(* Logix 5000 project; controller SX_V040001_C001 vendor 1 type 14 code 77 rev 16.23; software revision 16.04; part 30 of 35 *)
(* tags used below, declared in another part *)
   ALL_KINDS : INT[90];
   Basic : INT;
   DRIVE : INT[32];
   DRIVE_INTERVAL : INT[8];
   EMPTYING : INT[18];
   loading : INT[19];
   METERING : INT[44];
   NOTDOS : INT[6];
   pointer_recipe : DINT;
   pointer_recipe_line : DINT;
   pointer_recipe_restart : DINT;
   pointer_recipe_test : DINT;
   RECIPE_GENERAL : INT[405];
   T_MIN_ACTION_TIME : TIMER;
   TEMP : INT[14];
(* MainProgram, continued *)

ROUTINE RecipeRestart   (* ladder *)
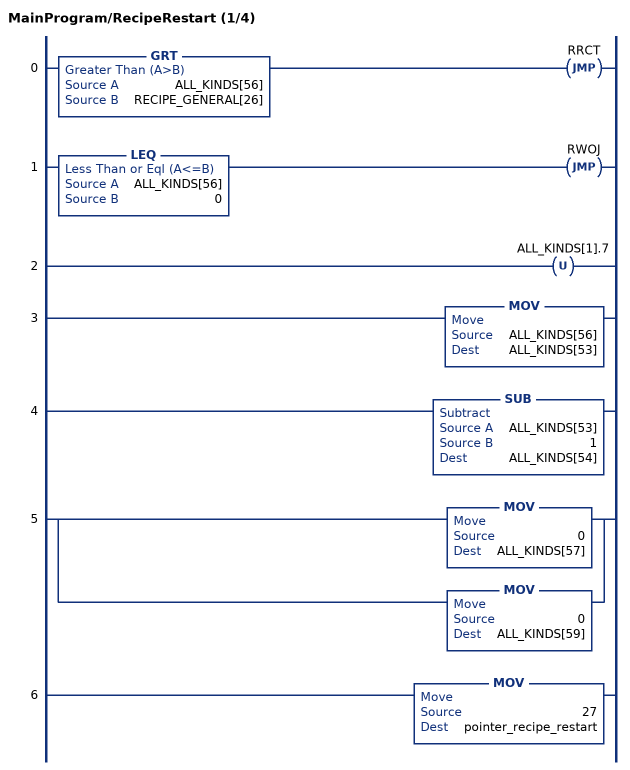
   0: GRT(ALL_KINDS[56],RECIPE_GENERAL[26])JMP(RRCT);
   1: LEQ(ALL_KINDS[56],0)JMP(RWOJ);
   2: OTU(ALL_KINDS[1].7);
   3: MOV(ALL_KINDS[56],ALL_KINDS[53]);
   4: SUB(ALL_KINDS[53],1,ALL_KINDS[54]);
   5: [MOV(0,ALL_KINDS[57]) ,MOV(0,ALL_KINDS[59]) ];
   6: MOV(27,pointer_recipe_restart);
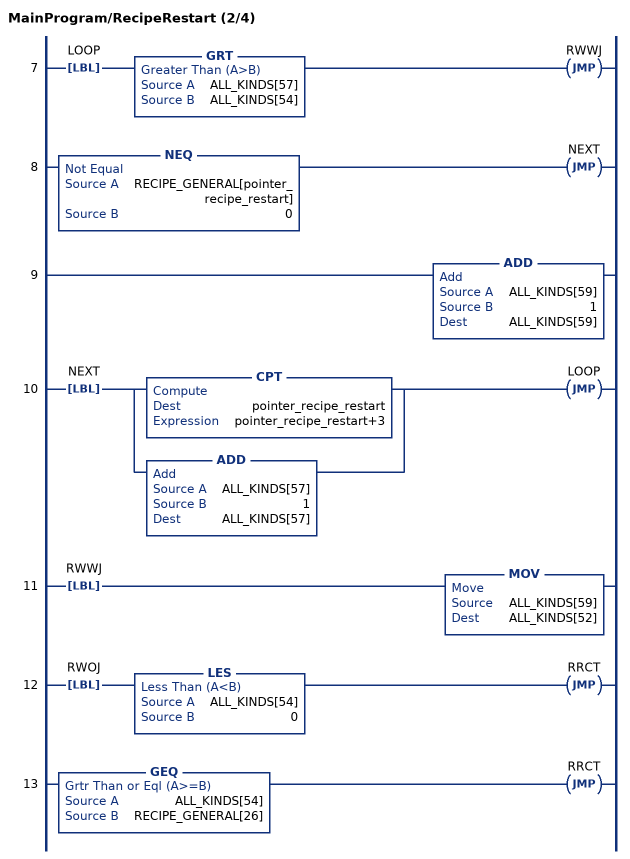
   7: LBL(LOOP)GRT(ALL_KINDS[57],ALL_KINDS[54])JMP(RWWJ);
   8: NEQ(RECIPE_GENERAL[pointer_recipe_restart],0)JMP(NEXT);
   9: ADD(ALL_KINDS[59],1,ALL_KINDS[59]);
   10: LBL(NEXT)[CPT(pointer_recipe_restart,pointer_recipe_restart+3) ,ADD(ALL_KINDS[57],1,ALL_KINDS[57]) ]JMP(LOOP);
   11: LBL(RWWJ)MOV(ALL_KINDS[59],ALL_KINDS[52]);
   12: LBL(RWOJ)LES(ALL_KINDS[54],0)JMP(RRCT);
   13: GEQ(ALL_KINDS[54],RECIPE_GENERAL[26])JMP(RRCT);
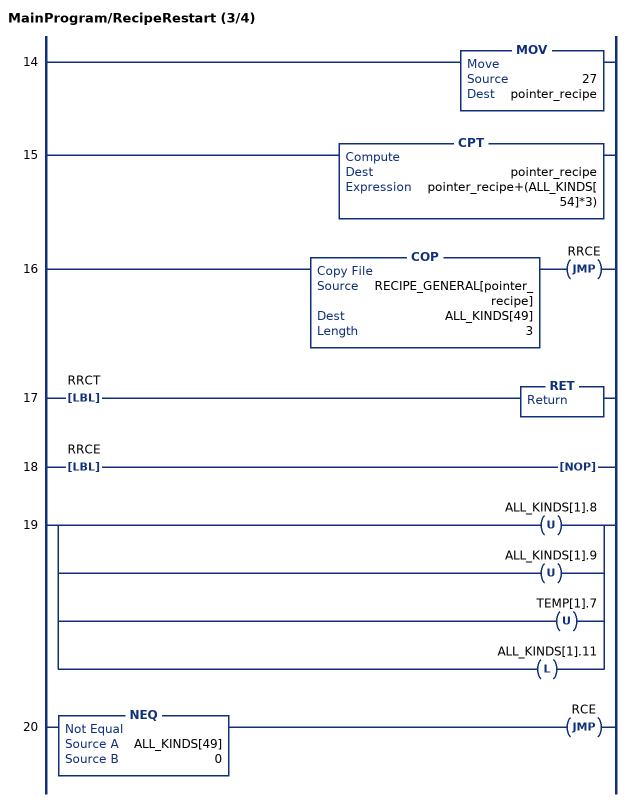
   14: MOV(27,pointer_recipe);
   15: CPT(pointer_recipe,pointer_recipe+(ALL_KINDS[54]*3));
   16: COP(RECIPE_GENERAL[pointer_recipe],ALL_KINDS[49],3)JMP(RRCE);
   17: LBL(RRCT)RET();
   18: LBL(RRCE)NOP();
   19: [OTU(ALL_KINDS[1].8) ,OTU(ALL_KINDS[1].9) ,OTU(TEMP[1].7) ,OTL(ALL_KINDS[1].11) ];
   20: NEQ(ALL_KINDS[49],0)JMP(RCE);
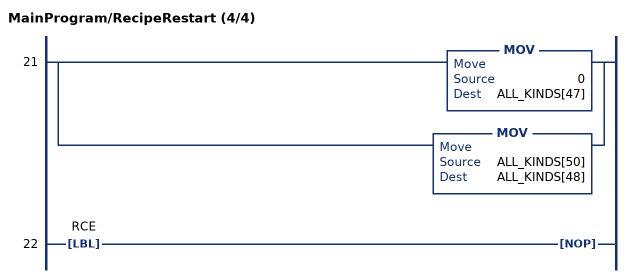
   21: [MOV(0,ALL_KINDS[47]) ,MOV(ALL_KINDS[50],ALL_KINDS[48]) ];
   22: LBL(RCE)NOP();
END_ROUTINE

ROUTINE RecipeRunning   (* ladder *)
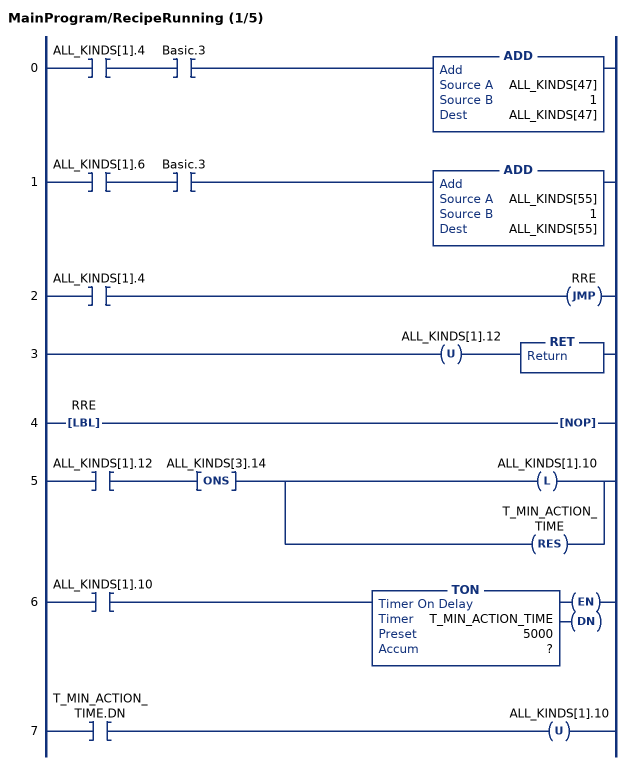
   0: XIC(ALL_KINDS[1].4)XIC(Basic.3)ADD(ALL_KINDS[47],1,ALL_KINDS[47]);
   1: XIC(ALL_KINDS[1].6)XIC(Basic.3)ADD(ALL_KINDS[55],1,ALL_KINDS[55]);
   2: XIC(ALL_KINDS[1].4)JMP(RRE);
   3: OTU(ALL_KINDS[1].12)RET();
   4: LBL(RRE)NOP();
   5: XIC(ALL_KINDS[1].12)ONS(ALL_KINDS[3].14)[OTL(ALL_KINDS[1].10) ,RES(T_MIN_ACTION_TIME) ];
   6: XIC(ALL_KINDS[1].10)TON(T_MIN_ACTION_TIME,?,?);
   7: XIC(T_MIN_ACTION_TIME.DN)OTU(ALL_KINDS[1].10);
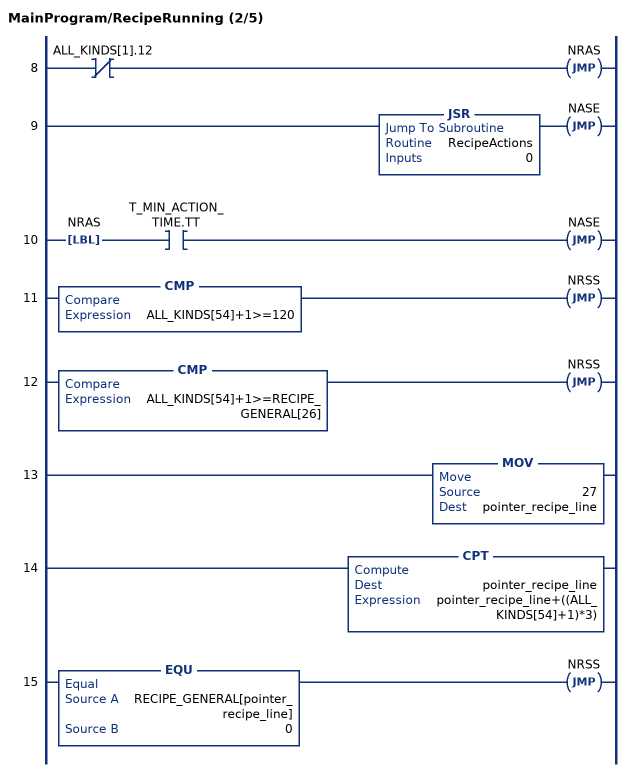
   8: XIO(ALL_KINDS[1].12)JMP(NRAS);
   9: JSR(RecipeActions,0)JMP(NASE);
   10: LBL(NRAS)XIC(T_MIN_ACTION_TIME.TT)JMP(NASE);
   11: CMP(ALL_KINDS[54]+1>=120)JMP(NRSS);
   12: CMP(ALL_KINDS[54]+1>=RECIPE_GENERAL[26])JMP(NRSS);
   13: MOV(27,pointer_recipe_line);
   14: CPT(pointer_recipe_line,pointer_recipe_line+((ALL_KINDS[54]+1)*3));
   15: EQU(RECIPE_GENERAL[pointer_recipe_line],0)JMP(NRSS);
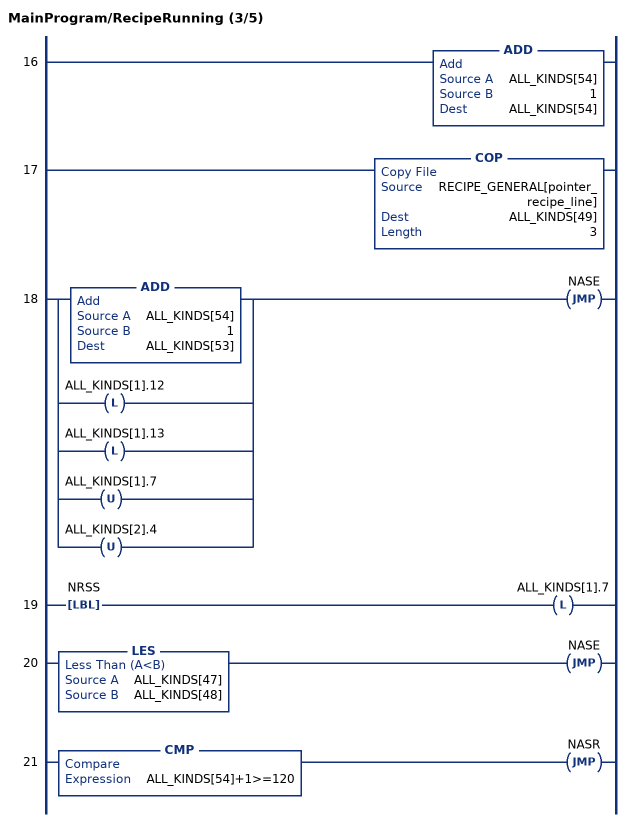
   16: ADD(ALL_KINDS[54],1,ALL_KINDS[54]);
   17: COP(RECIPE_GENERAL[pointer_recipe_line],ALL_KINDS[49],3);
   18: [ADD(ALL_KINDS[54],1,ALL_KINDS[53]) ,OTL(ALL_KINDS[1].12) ,OTL(ALL_KINDS[1].13) ,OTU(ALL_KINDS[1].7) ,OTU(ALL_KINDS[2].4) ]JMP(NASE);
   19: LBL(NRSS)OTL(ALL_KINDS[1].7);
   20: LES(ALL_KINDS[47],ALL_KINDS[48])JMP(NASE);
   21: CMP(ALL_KINDS[54]+1>=120)JMP(NASR);
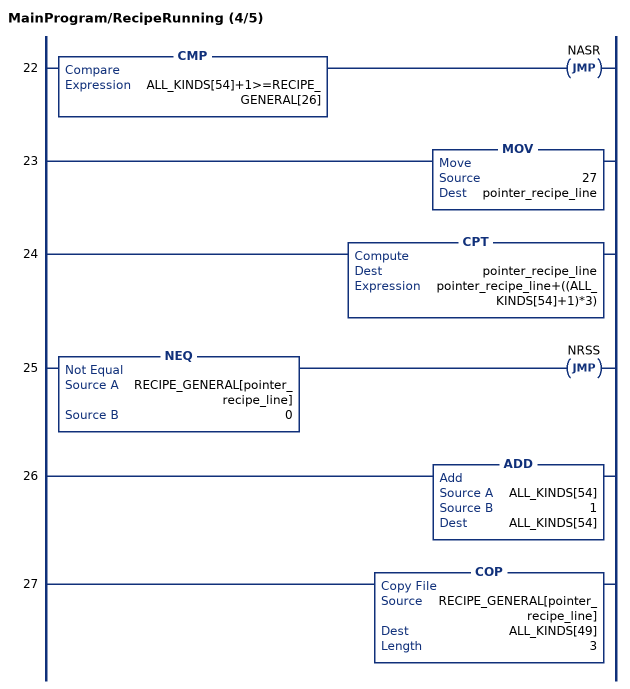
   22: CMP(ALL_KINDS[54]+1>=RECIPE_GENERAL[26])JMP(NASR);
   23: MOV(27,pointer_recipe_line);
   24: CPT(pointer_recipe_line,pointer_recipe_line+((ALL_KINDS[54]+1)*3));
   25: NEQ(RECIPE_GENERAL[pointer_recipe_line],0)JMP(NRSS);
   26: ADD(ALL_KINDS[54],1,ALL_KINDS[54]);
   27: COP(RECIPE_GENERAL[pointer_recipe_line],ALL_KINDS[49],3);
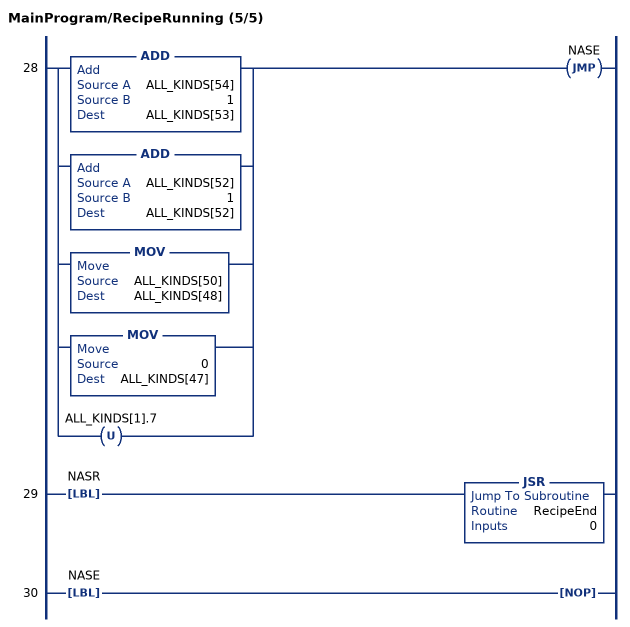
   28: [ADD(ALL_KINDS[54],1,ALL_KINDS[53]) ,ADD(ALL_KINDS[52],1,ALL_KINDS[52]) ,MOV(ALL_KINDS[50],ALL_KINDS[48]) ,MOV(0,ALL_KINDS[47]) ,OTU(ALL_KINDS[1].7) ]JMP(NASE);
   29: LBL(NASR)JSR(RecipeEnd,0);
   30: LBL(NASE)NOP();
END_ROUTINE

ROUTINE RecipeTermination   (* ladder *)
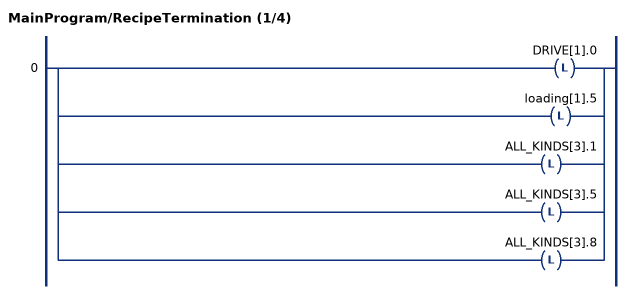
   0: [OTL(DRIVE[1].0) ,OTL(loading[1].5) ,OTL(ALL_KINDS[3].1) ,OTL(ALL_KINDS[3].5) ,OTL(ALL_KINDS[3].8) ];
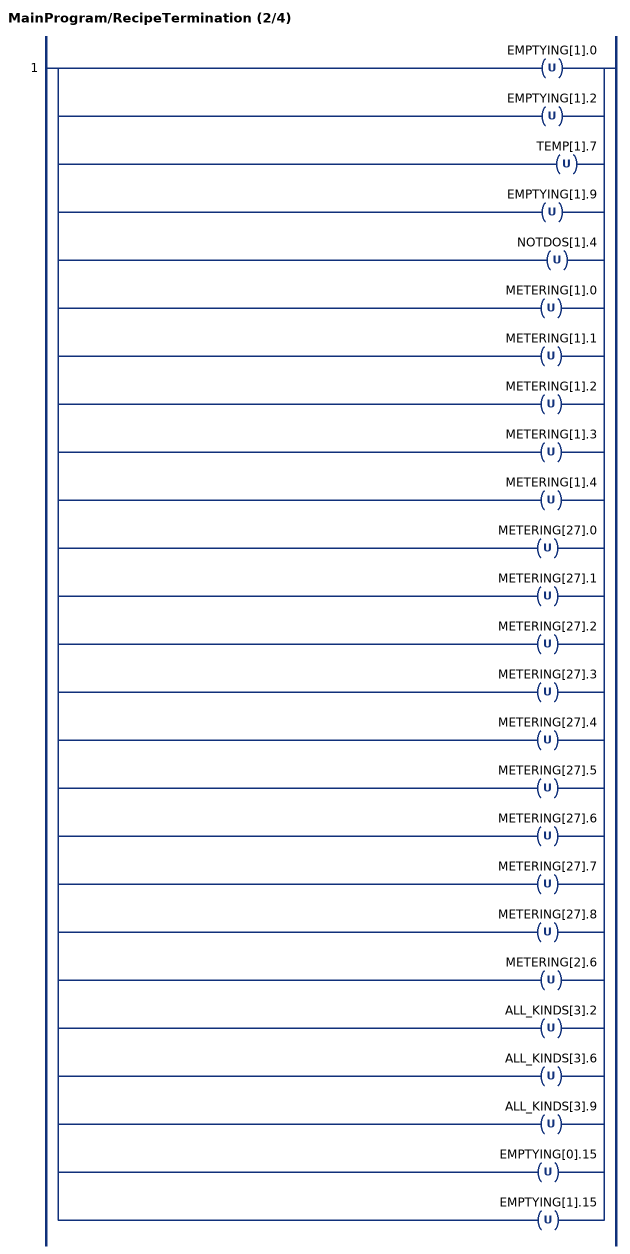
   1: [OTU(EMPTYING[1].0) ,OTU(EMPTYING[1].2) ,OTU(TEMP[1].7) ,OTU(EMPTYING[1].9) ,OTU(NOTDOS[1].4) ,OTU(METERING[1].0) ,OTU(METERING[1].1) ,OTU(METERING[1].2) ,OTU(METERING[1].3) ,OTU(METERING[1].4) ,OTU(METERING[27].0) ,OTU(METERING[27].1) ,OTU(METERING[27].2) ,OTU(METERING[27].3) ,OTU(METERING[27].4) ,OTU(METERING[27].5) ,OTU(METERING[27].6) ,OTU(METERING[27].7) ,OTU(METERING[27].8) ,OTU(METERING[2].6) ,OTU(ALL_KINDS[3].2) ,OTU(ALL_KINDS[3].6) ,OTU(ALL_KINDS[3].9) ,OTU(EMPTYING[0].15) ,OTU(EMPTYING[1].15) ];
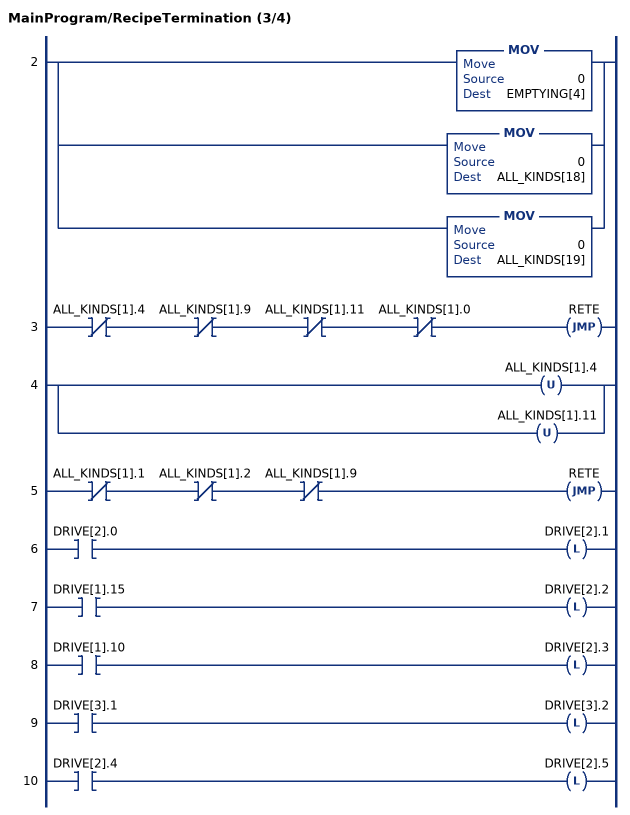
   2: [MOV(0,EMPTYING[4]) ,MOV(0,ALL_KINDS[18]) ,MOV(0,ALL_KINDS[19]) ];
   3: XIO(ALL_KINDS[1].4)XIO(ALL_KINDS[1].9)XIO(ALL_KINDS[1].11)XIO(ALL_KINDS[1].0)JMP(RETE);
   4: [OTU(ALL_KINDS[1].4) ,OTU(ALL_KINDS[1].11) ];
   5: XIO(ALL_KINDS[1].1)XIO(ALL_KINDS[1].2)XIO(ALL_KINDS[1].9)JMP(RETE);
   6: XIC(DRIVE[2].0)OTL(DRIVE[2].1);
   7: XIC(DRIVE[1].15)OTL(DRIVE[2].2);
   8: XIC(DRIVE[1].10)OTL(DRIVE[2].3);
   9: XIC(DRIVE[3].1)OTL(DRIVE[3].2);
   10: XIC(DRIVE[2].4)OTL(DRIVE[2].5);
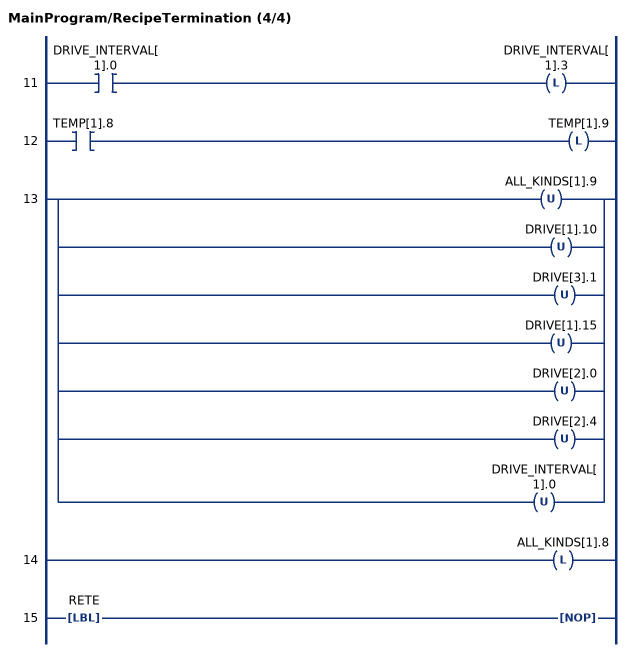
   11: XIC(DRIVE_INTERVAL[1].0)OTL(DRIVE_INTERVAL[1].3);
   12: XIC(TEMP[1].8)OTL(TEMP[1].9);
   13: [OTU(ALL_KINDS[1].9) ,OTU(DRIVE[1].10) ,OTU(DRIVE[3].1) ,OTU(DRIVE[1].15) ,OTU(DRIVE[2].0) ,OTU(DRIVE[2].4) ,OTU(DRIVE_INTERVAL[1].0) ];
   14: OTL(ALL_KINDS[1].8);
   15: LBL(RETE)NOP();
END_ROUTINE

ROUTINE RecipeTest   (* ladder *)
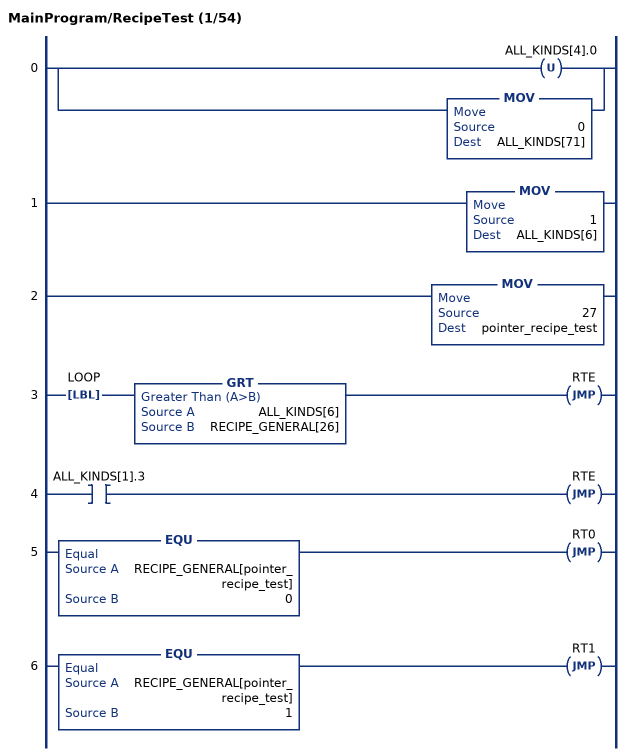
   0: [OTU(ALL_KINDS[4].0) ,MOV(0,ALL_KINDS[71]) ];
   1: MOV(1,ALL_KINDS[6]);
   2: MOV(27,pointer_recipe_test);
   3: LBL(LOOP)GRT(ALL_KINDS[6],RECIPE_GENERAL[26])JMP(RTE);
   4: XIC(ALL_KINDS[1].3)JMP(RTE);
   5: EQU(RECIPE_GENERAL[pointer_recipe_test],0)JMP(RT0);
   6: EQU(RECIPE_GENERAL[pointer_recipe_test],1)JMP(RT1);
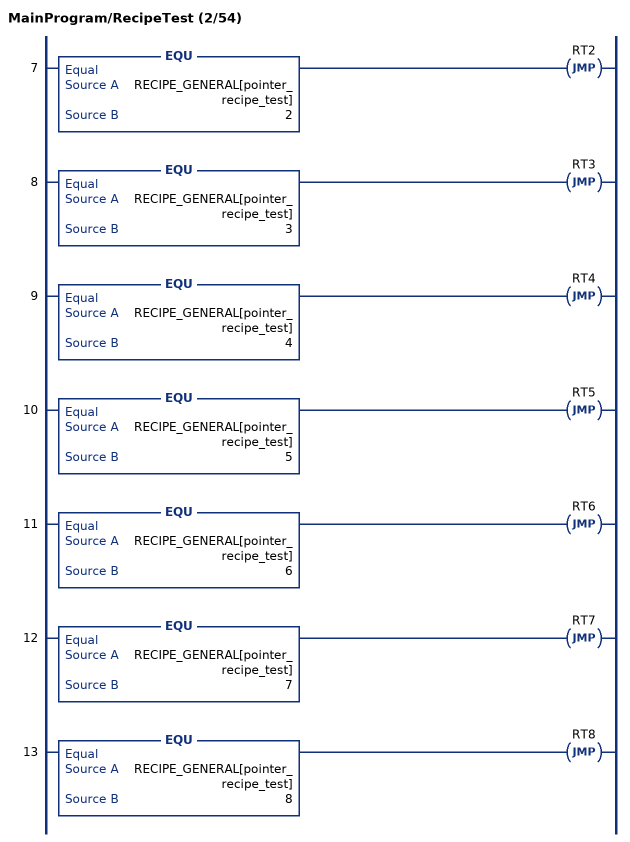
   7: EQU(RECIPE_GENERAL[pointer_recipe_test],2)JMP(RT2);
   8: EQU(RECIPE_GENERAL[pointer_recipe_test],3)JMP(RT3);
   9: EQU(RECIPE_GENERAL[pointer_recipe_test],4)JMP(RT4);
   10: EQU(RECIPE_GENERAL[pointer_recipe_test],5)JMP(RT5);
   11: EQU(RECIPE_GENERAL[pointer_recipe_test],6)JMP(RT6);
   12: EQU(RECIPE_GENERAL[pointer_recipe_test],7)JMP(RT7);
   13: EQU(RECIPE_GENERAL[pointer_recipe_test],8)JMP(RT8);
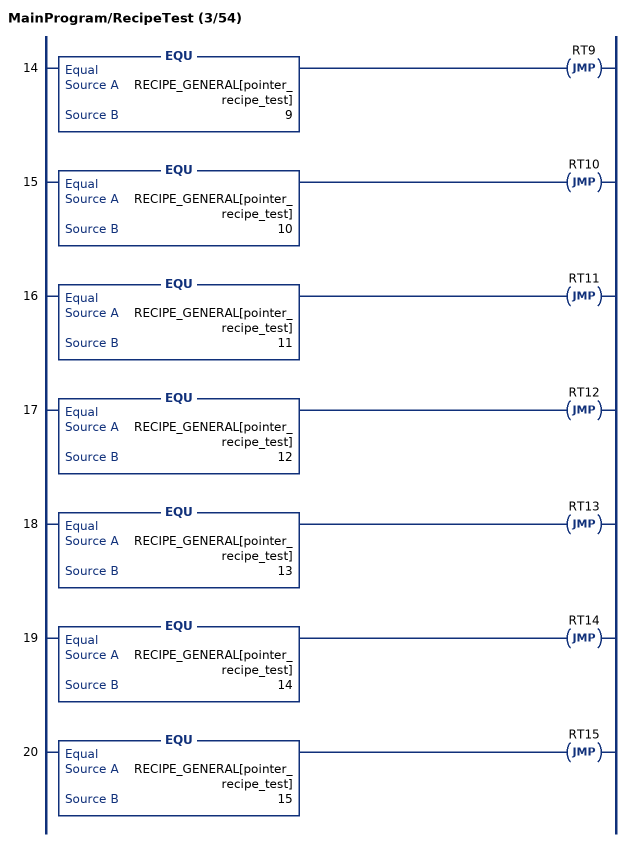
   14: EQU(RECIPE_GENERAL[pointer_recipe_test],9)JMP(RT9);
   15: EQU(RECIPE_GENERAL[pointer_recipe_test],10)JMP(RT10);
   16: EQU(RECIPE_GENERAL[pointer_recipe_test],11)JMP(RT11);
   17: EQU(RECIPE_GENERAL[pointer_recipe_test],12)JMP(RT12);
   18: EQU(RECIPE_GENERAL[pointer_recipe_test],13)JMP(RT13);
   19: EQU(RECIPE_GENERAL[pointer_recipe_test],14)JMP(RT14);
   20: EQU(RECIPE_GENERAL[pointer_recipe_test],15)JMP(RT15);
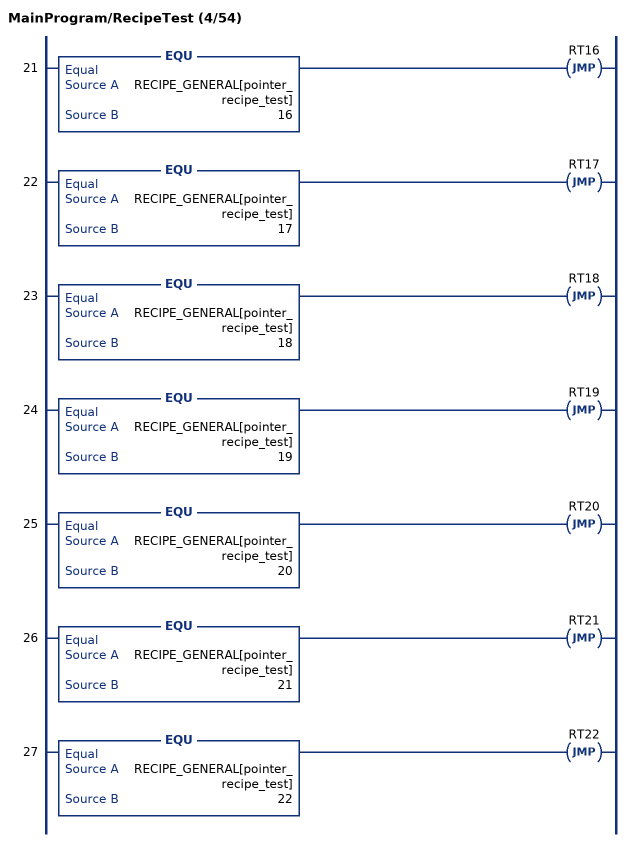
   21: EQU(RECIPE_GENERAL[pointer_recipe_test],16)JMP(RT16);
   22: EQU(RECIPE_GENERAL[pointer_recipe_test],17)JMP(RT17);
   23: EQU(RECIPE_GENERAL[pointer_recipe_test],18)JMP(RT18);
   24: EQU(RECIPE_GENERAL[pointer_recipe_test],19)JMP(RT19);
   25: EQU(RECIPE_GENERAL[pointer_recipe_test],20)JMP(RT20);
   26: EQU(RECIPE_GENERAL[pointer_recipe_test],21)JMP(RT21);
   27: EQU(RECIPE_GENERAL[pointer_recipe_test],22)JMP(RT22);
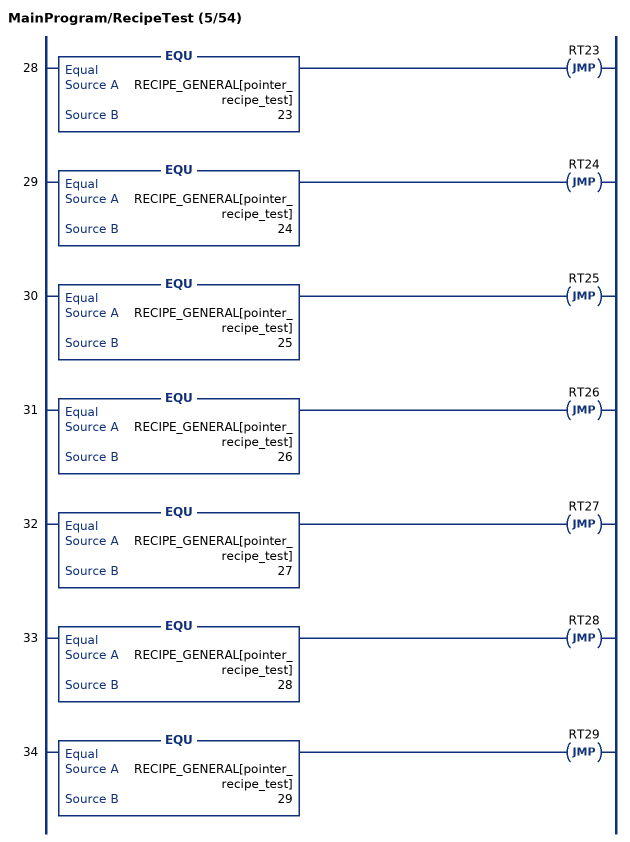
   28: EQU(RECIPE_GENERAL[pointer_recipe_test],23)JMP(RT23);
   29: EQU(RECIPE_GENERAL[pointer_recipe_test],24)JMP(RT24);
   30: EQU(RECIPE_GENERAL[pointer_recipe_test],25)JMP(RT25);
   31: EQU(RECIPE_GENERAL[pointer_recipe_test],26)JMP(RT26);
   32: EQU(RECIPE_GENERAL[pointer_recipe_test],27)JMP(RT27);
   33: EQU(RECIPE_GENERAL[pointer_recipe_test],28)JMP(RT28);
   34: EQU(RECIPE_GENERAL[pointer_recipe_test],29)JMP(RT29);
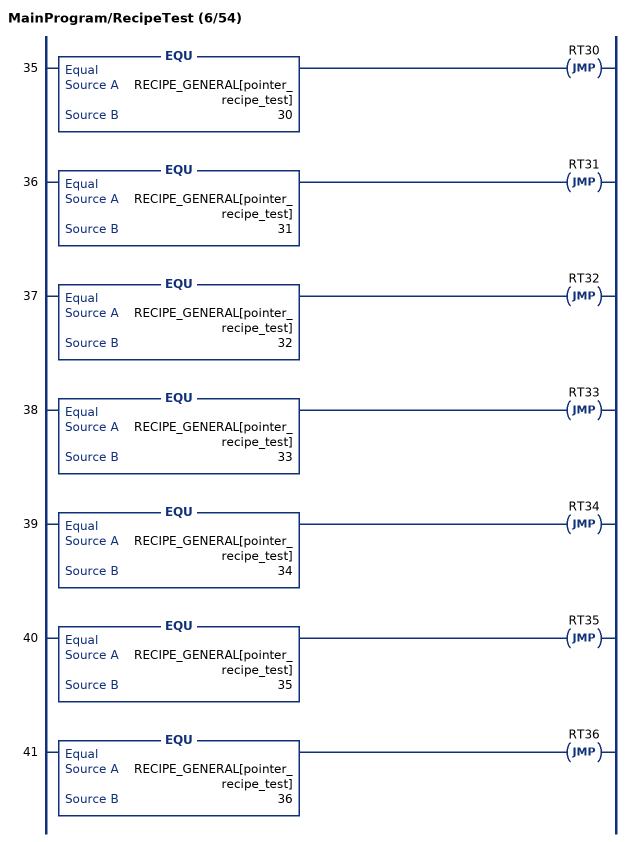
   35: EQU(RECIPE_GENERAL[pointer_recipe_test],30)JMP(RT30);
   36: EQU(RECIPE_GENERAL[pointer_recipe_test],31)JMP(RT31);
   37: EQU(RECIPE_GENERAL[pointer_recipe_test],32)JMP(RT32);
   38: EQU(RECIPE_GENERAL[pointer_recipe_test],33)JMP(RT33);
   39: EQU(RECIPE_GENERAL[pointer_recipe_test],34)JMP(RT34);
   40: EQU(RECIPE_GENERAL[pointer_recipe_test],35)JMP(RT35);
   41: EQU(RECIPE_GENERAL[pointer_recipe_test],36)JMP(RT36);
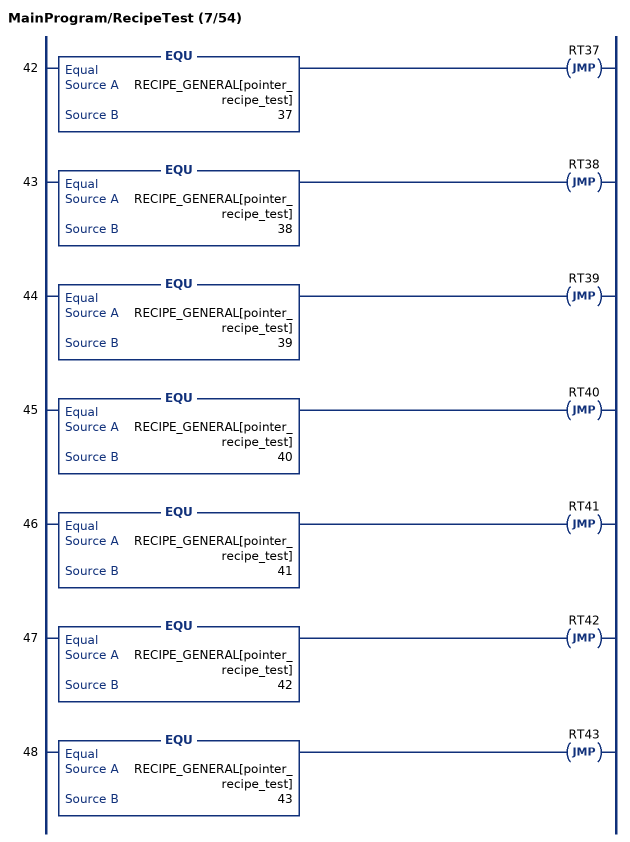
   42: EQU(RECIPE_GENERAL[pointer_recipe_test],37)JMP(RT37);
   43: EQU(RECIPE_GENERAL[pointer_recipe_test],38)JMP(RT38);
   44: EQU(RECIPE_GENERAL[pointer_recipe_test],39)JMP(RT39);
   45: EQU(RECIPE_GENERAL[pointer_recipe_test],40)JMP(RT40);
   46: EQU(RECIPE_GENERAL[pointer_recipe_test],41)JMP(RT41);
   47: EQU(RECIPE_GENERAL[pointer_recipe_test],42)JMP(RT42);
   48: EQU(RECIPE_GENERAL[pointer_recipe_test],43)JMP(RT43);
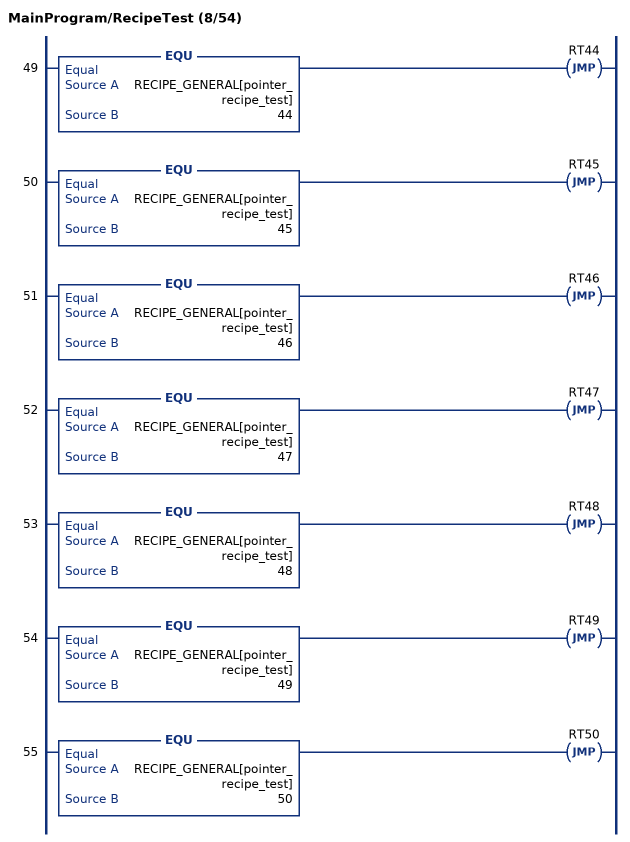
   49: EQU(RECIPE_GENERAL[pointer_recipe_test],44)JMP(RT44);
   50: EQU(RECIPE_GENERAL[pointer_recipe_test],45)JMP(RT45);
   51: EQU(RECIPE_GENERAL[pointer_recipe_test],46)JMP(RT46);
   52: EQU(RECIPE_GENERAL[pointer_recipe_test],47)JMP(RT47);
   53: EQU(RECIPE_GENERAL[pointer_recipe_test],48)JMP(RT48);
   54: EQU(RECIPE_GENERAL[pointer_recipe_test],49)JMP(RT49);
   55: EQU(RECIPE_GENERAL[pointer_recipe_test],50)JMP(RT50);
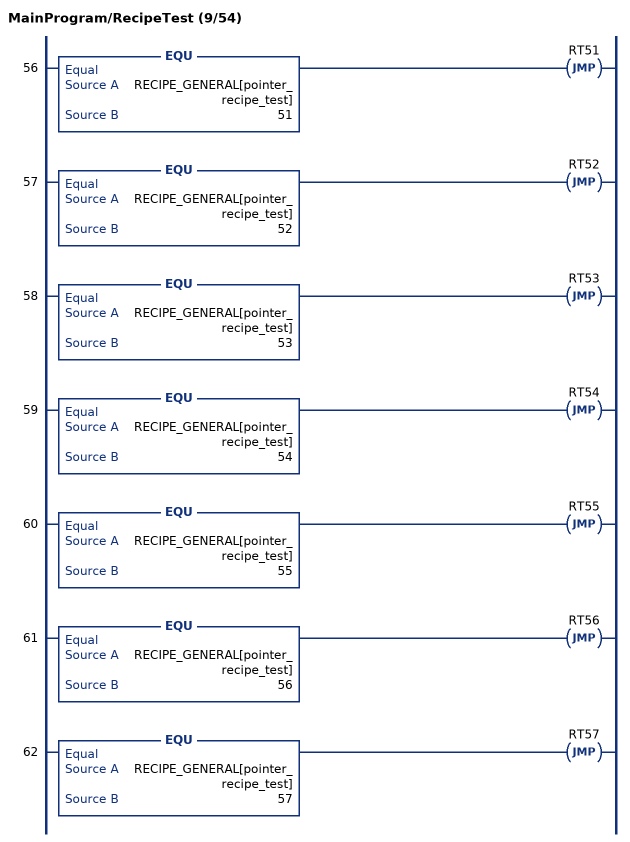
   56: EQU(RECIPE_GENERAL[pointer_recipe_test],51)JMP(RT51);
   57: EQU(RECIPE_GENERAL[pointer_recipe_test],52)JMP(RT52);
   58: EQU(RECIPE_GENERAL[pointer_recipe_test],53)JMP(RT53);
   59: EQU(RECIPE_GENERAL[pointer_recipe_test],54)JMP(RT54);
   60: EQU(RECIPE_GENERAL[pointer_recipe_test],55)JMP(RT55);
   61: EQU(RECIPE_GENERAL[pointer_recipe_test],56)JMP(RT56);
   62: EQU(RECIPE_GENERAL[pointer_recipe_test],57)JMP(RT57);
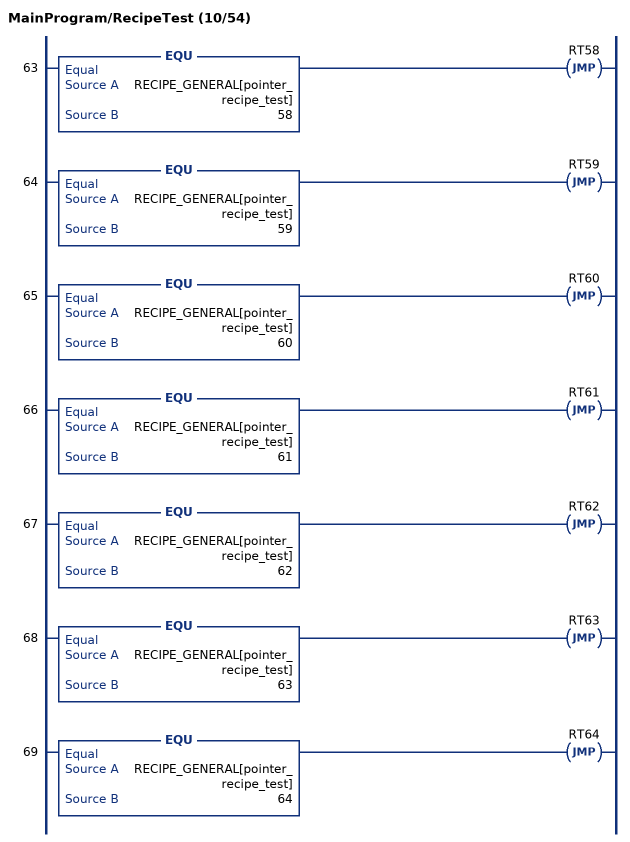
   63: EQU(RECIPE_GENERAL[pointer_recipe_test],58)JMP(RT58);
   64: EQU(RECIPE_GENERAL[pointer_recipe_test],59)JMP(RT59);
   65: EQU(RECIPE_GENERAL[pointer_recipe_test],60)JMP(RT60);
   66: EQU(RECIPE_GENERAL[pointer_recipe_test],61)JMP(RT61);
   67: EQU(RECIPE_GENERAL[pointer_recipe_test],62)JMP(RT62);
   68: EQU(RECIPE_GENERAL[pointer_recipe_test],63)JMP(RT63);
   69: EQU(RECIPE_GENERAL[pointer_recipe_test],64)JMP(RT64);
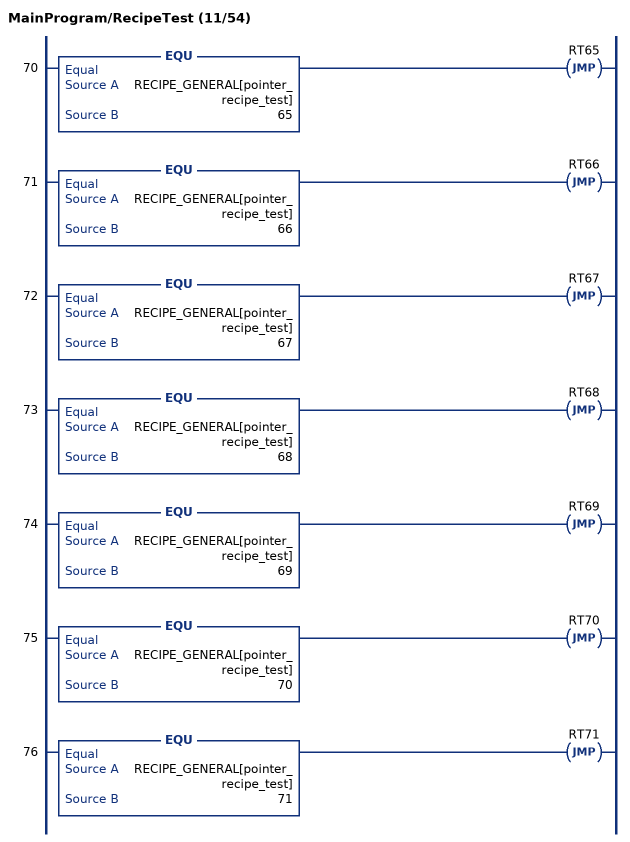
   70: EQU(RECIPE_GENERAL[pointer_recipe_test],65)JMP(RT65);
   71: EQU(RECIPE_GENERAL[pointer_recipe_test],66)JMP(RT66);
   72: EQU(RECIPE_GENERAL[pointer_recipe_test],67)JMP(RT67);
   73: EQU(RECIPE_GENERAL[pointer_recipe_test],68)JMP(RT68);
   74: EQU(RECIPE_GENERAL[pointer_recipe_test],69)JMP(RT69);
   75: EQU(RECIPE_GENERAL[pointer_recipe_test],70)JMP(RT70);
   76: EQU(RECIPE_GENERAL[pointer_recipe_test],71)JMP(RT71);
